// TIA Portal V20 export
FUNCTION_BLOCK "FB_Msg"   // FB84, SCL
{ S7_Optimized_Access := 'TRUE' }
// stored: MemoryReserve 100, SetENOAutomatically false
   VAR
      sSeverity : Byte;
      sMemoNumberOfActiveAlarms : DInt;
      sTON_On : TON_TIME;
      sTON_OFF { S7_SetPoint := 'True'} : TON_TIME;
      sPulseUpdateAlarms { S7_SetPoint := 'True'} : Bool;
      sRT_PulseUpdateAlarms : R_TRIG;
   END_VAR
   VAR_TEMP
      tIndex1 : Int;
      tIndex2 : Int;
      tResultByte0 : Int;
   END_VAR
   VAR CONSTANT
      MSG_SIZE : Int := 95;
   END_VAR
BEGIN
   // REGION Test
   //     FOR #tIndex := 0 TO #MSG_SIZE DO
   //         #tResultByte0 := PEEK(area := 16#84, dbNumber := 2, byteOffset := #tIndex + 554);
   //         "Db_Messages".Msg[#tIndex].ID := #tIndex;
   //         "Db_Messages".Msg[#tIndex].Number := INT_TO_DINT(#tIndex) + 70000;
   //         "Db_Messages".Msg[#tIndex].Active := #tResultByte0.%X0;
   //     END_FOR;
   // END_REGION

   REGION Format Msg
       // Mise en forme des alarmes (DB2) dans DB_FormatMsg
       FOR #tIndex1 := 0 TO 8 DO
           FOR #tIndex2 := 0 TO 7 DO
               #tResultByte0 := PEEK(area := 16#84, dbNumber := 2, byteOffset := #tIndex2 + 554 + (#tIndex1 * 8));
               "DB_FormatMsg".Msg[(#tIndex2 * 8) + (#tIndex1 * 64) + 0].Id := INT_TO_DINT((#tIndex2 * 8) + 0) + 70000 + (#tIndex1 * 100);
               "DB_FormatMsg".Msg[(#tIndex2 * 8) + (#tIndex1 * 64) + 1].Id := INT_TO_DINT((#tIndex2 * 8) + 1) + 70000 + (#tIndex1 * 100);
               "DB_FormatMsg".Msg[(#tIndex2 * 8) + (#tIndex1 * 64) + 2].Id := INT_TO_DINT((#tIndex2 * 8) + 2) + 70000 + (#tIndex1 * 100);
               "DB_FormatMsg".Msg[(#tIndex2 * 8) + (#tIndex1 * 64) + 3].Id := INT_TO_DINT((#tIndex2 * 8) + 3) + 70000 + (#tIndex1 * 100);
               "DB_FormatMsg".Msg[(#tIndex2 * 8) + (#tIndex1 * 64) + 4].Id := INT_TO_DINT((#tIndex2 * 8) + 4) + 70000 + (#tIndex1 * 100);
               "DB_FormatMsg".Msg[(#tIndex2 * 8) + (#tIndex1 * 64) + 5].Id := INT_TO_DINT((#tIndex2 * 8) + 5) + 70000 + (#tIndex1 * 100);
               "DB_FormatMsg".Msg[(#tIndex2 * 8) + (#tIndex1 * 64) + 6].Id := INT_TO_DINT((#tIndex2 * 8) + 6) + 70000 + (#tIndex1 * 100);
               "DB_FormatMsg".Msg[(#tIndex2 * 8) + (#tIndex1 * 64) + 7].Id := INT_TO_DINT((#tIndex2 * 8) + 7) + 70000 + (#tIndex1 * 100);

               "DB_FormatMsg".Msg[(#tIndex2 * 8) + (#tIndex1 * 64) + 0].Active := #tResultByte0.%X0;
               "DB_FormatMsg".Msg[(#tIndex2 * 8) + (#tIndex1 * 64) + 1].Active := #tResultByte0.%X1;
               "DB_FormatMsg".Msg[(#tIndex2 * 8) + (#tIndex1 * 64) + 2].Active := #tResultByte0.%X2;
               "DB_FormatMsg".Msg[(#tIndex2 * 8) + (#tIndex1 * 64) + 3].Active := #tResultByte0.%X3;
               "DB_FormatMsg".Msg[(#tIndex2 * 8) + (#tIndex1 * 64) + 4].Active := #tResultByte0.%X4;
               "DB_FormatMsg".Msg[(#tIndex2 * 8) + (#tIndex1 * 64) + 5].Active := #tResultByte0.%X5;
               "DB_FormatMsg".Msg[(#tIndex2 * 8) + (#tIndex1 * 64) + 6].Active := #tResultByte0.%X6;
               "DB_FormatMsg".Msg[(#tIndex2 * 8) + (#tIndex1 * 64) + 7].Active := #tResultByte0.%X7;
           END_FOR;
       END_FOR;
   END_REGION

   REGION Severity WFA A REVOIR !!
       #sSeverity := 1;
       "DB_FormatMsg".Msg[35].Severity := #sSeverity;

       "DB_FormatMsg".Msg[236].Severity := #sSeverity;

       "DB_FormatMsg".Msg[532].Severity := #sSeverity;
       "DB_FormatMsg".Msg[533].Severity := #sSeverity;
       "DB_FormatMsg".Msg[534].Severity := #sSeverity;
       "DB_FormatMsg".Msg[535].Severity := #sSeverity;
       "DB_FormatMsg".Msg[536].Severity := #sSeverity;
       "DB_FormatMsg".Msg[537].Severity := #sSeverity;
       "DB_FormatMsg".Msg[538].Severity := #sSeverity;
       "DB_FormatMsg".Msg[539].Severity := #sSeverity;
       "DB_FormatMsg".Msg[542].Severity := #sSeverity;
       "DB_FormatMsg".Msg[548].Severity := #sSeverity;
       "DB_FormatMsg".Msg[550].Severity := #sSeverity;
       "DB_FormatMsg".Msg[551].Severity := #sSeverity;

       "DB_FormatMsg".Msg[800].Severity := #sSeverity;
       "DB_FormatMsg".Msg[841].Severity := #sSeverity;

       #sSeverity := 2;
       "DB_FormatMsg".Msg[59].Severity := #sSeverity;
       "DB_FormatMsg".Msg[60].Severity := #sSeverity;
       "DB_FormatMsg".Msg[61].Severity := #sSeverity;
       "DB_FormatMsg".Msg[62].Severity := #sSeverity;

       "DB_FormatMsg".Msg[348].Severity := #sSeverity;

       "DB_FormatMsg".Msg[441].Severity := #sSeverity;
       "DB_FormatMsg".Msg[442].Severity := #sSeverity;

       "DB_FormatMsg".Msg[543].Severity := #sSeverity;

       "DB_FormatMsg".Msg[662].Severity := #sSeverity;
       "DB_FormatMsg".Msg[663].Severity := #sSeverity;

       // "DB_FormatMsg".Msg[3032].Severity := #sSeverity;
       // "DB_FormatMsg".Msg[3033].Severity := #sSeverity;
       // "DB_FormatMsg".Msg[3034].Severity := #sSeverity;
       // "DB_FormatMsg".Msg[3035].Severity := #sSeverity;
       // "DB_FormatMsg".Msg[3036].Severity := #sSeverity;
       // "DB_FormatMsg".Msg[3037].Severity := #sSeverity;
       // "DB_FormatMsg".Msg[3038].Severity := #sSeverity;
       // "DB_FormatMsg".Msg[3039].Severity := #sSeverity;
       // "DB_FormatMsg".Msg[3010].Severity := #sSeverity;
       // "DB_FormatMsg".Msg[3041].Severity := #sSeverity;
       // "DB_FormatMsg".Msg[3042].Severity := #sSeverity;
       // "DB_FormatMsg".Msg[3043].Severity := #sSeverity;
       // "DB_FormatMsg".Msg[3044].Severity := #sSeverity;
       // "DB_FormatMsg".Msg[3045].Severity := #sSeverity;
       // "DB_FormatMsg".Msg[3046].Severity := #sSeverity;
       // "DB_FormatMsg".Msg[3047].Severity := #sSeverity;


       "DB_FormatMsg".Msg[55].Severity := #sSeverity;
       "DB_FormatMsg".Msg[63].Severity := #sSeverity;

       "DB_FormatMsg".Msg[403].Severity := #sSeverity;
       "DB_FormatMsg".Msg[404].Severity := #sSeverity;
       "DB_FormatMsg".Msg[405].Severity := #sSeverity;
       "DB_FormatMsg".Msg[406].Severity := #sSeverity;
       "DB_FormatMsg".Msg[420].Severity := #sSeverity;
       "DB_FormatMsg".Msg[421].Severity := #sSeverity;
       "DB_FormatMsg".Msg[422].Severity := #sSeverity;
       "DB_FormatMsg".Msg[423].Severity := #sSeverity;

       "DB_FormatMsg".Msg[508].Severity := #sSeverity;
       "DB_FormatMsg".Msg[509].Severity := #sSeverity;
       "DB_FormatMsg".Msg[510].Severity := #sSeverity;
       "DB_FormatMsg".Msg[511].Severity := #sSeverity;
       "DB_FormatMsg".Msg[512].Severity := #sSeverity;

       "DB_FormatMsg".Msg[652].Severity := #sSeverity;
       "DB_FormatMsg".Msg[653].Severity := #sSeverity;

       "DB_FormatMsg".Msg[700].Severity := #sSeverity;
       "DB_FormatMsg".Msg[701].Severity := #sSeverity;
       "DB_FormatMsg".Msg[702].Severity := #sSeverity;
       "DB_FormatMsg".Msg[703].Severity := #sSeverity;
       "DB_FormatMsg".Msg[704].Severity := #sSeverity;
       "DB_FormatMsg".Msg[705].Severity := #sSeverity;
       "DB_FormatMsg".Msg[706].Severity := #sSeverity;
       "DB_FormatMsg".Msg[707].Severity := #sSeverity;
       "DB_FormatMsg".Msg[708].Severity := #sSeverity;
       "DB_FormatMsg".Msg[709].Severity := #sSeverity;
       "DB_FormatMsg".Msg[710].Severity := #sSeverity;
       "DB_FormatMsg".Msg[711].Severity := #sSeverity;
       "DB_FormatMsg".Msg[740].Severity := #sSeverity;
       "DB_FormatMsg".Msg[741].Severity := #sSeverity;
       "DB_FormatMsg".Msg[742].Severity := #sSeverity;
       "DB_FormatMsg".Msg[743].Severity := #sSeverity;
       "DB_FormatMsg".Msg[744].Severity := #sSeverity;
       "DB_FormatMsg".Msg[745].Severity := #sSeverity;
       "DB_FormatMsg".Msg[746].Severity := #sSeverity;
       "DB_FormatMsg".Msg[747].Severity := #sSeverity;
       "DB_FormatMsg".Msg[748].Severity := #sSeverity;
       "DB_FormatMsg".Msg[749].Severity := #sSeverity;
       "DB_FormatMsg".Msg[750].Severity := #sSeverity;
       "DB_FormatMsg".Msg[751].Severity := #sSeverity;
       "DB_FormatMsg".Msg[752].Severity := #sSeverity;
       "DB_FormatMsg".Msg[753].Severity := #sSeverity;
       "DB_FormatMsg".Msg[754].Severity := #sSeverity;
       "DB_FormatMsg".Msg[755].Severity := #sSeverity;
       "DB_FormatMsg".Msg[756].Severity := #sSeverity;
       "DB_FormatMsg".Msg[757].Severity := #sSeverity;
       "DB_FormatMsg".Msg[758].Severity := #sSeverity;
       "DB_FormatMsg".Msg[759].Severity := #sSeverity;
       "DB_FormatMsg".Msg[760].Severity := #sSeverity;
       "DB_FormatMsg".Msg[761].Severity := #sSeverity;

       // "DB_FormatMsg".Msg[3000].Severity := #sSeverity;
       // "DB_FormatMsg".Msg[3001].Severity := #sSeverity;
       // "DB_FormatMsg".Msg[3002].Severity := #sSeverity;
       // "DB_FormatMsg".Msg[3003].Severity := #sSeverity;
       // "DB_FormatMsg".Msg[3004].Severity := #sSeverity;
       // "DB_FormatMsg".Msg[3005].Severity := #sSeverity;
       // "DB_FormatMsg".Msg[3006].Severity := #sSeverity;
       // "DB_FormatMsg".Msg[3007].Severity := #sSeverity;
       // "DB_FormatMsg".Msg[3008].Severity := #sSeverity;
       // "DB_FormatMsg".Msg[3009].Severity := #sSeverity;
       // "DB_FormatMsg".Msg[3010].Severity := #sSeverity;
       // "DB_FormatMsg".Msg[3011].Severity := #sSeverity;
       // "DB_FormatMsg".Msg[3012].Severity := #sSeverity;
       // "DB_FormatMsg".Msg[3013].Severity := #sSeverity;
       // "DB_FormatMsg".Msg[3014].Severity := #sSeverity;
       // "DB_FormatMsg".Msg[3015].Severity := #sSeverity;


       #sSeverity := 3;
       "DB_FormatMsg".Msg[6].Severity := #sSeverity;
       "DB_FormatMsg".Msg[7].Severity := #sSeverity;
       "DB_FormatMsg".Msg[8].Severity := #sSeverity;

       "DB_FormatMsg".Msg[103].Severity := #sSeverity;
       "DB_FormatMsg".Msg[104].Severity := #sSeverity;
       "DB_FormatMsg".Msg[105].Severity := #sSeverity;
       "DB_FormatMsg".Msg[106].Severity := #sSeverity;
       "DB_FormatMsg".Msg[107].Severity := #sSeverity;
       "DB_FormatMsg".Msg[108].Severity := #sSeverity;
       "DB_FormatMsg".Msg[109].Severity := #sSeverity;
       "DB_FormatMsg".Msg[110].Severity := #sSeverity;
       "DB_FormatMsg".Msg[111].Severity := #sSeverity;
       "DB_FormatMsg".Msg[112].Severity := #sSeverity;
       "DB_FormatMsg".Msg[113].Severity := #sSeverity;
       "DB_FormatMsg".Msg[114].Severity := #sSeverity;
       "DB_FormatMsg".Msg[115].Severity := #sSeverity;
       "DB_FormatMsg".Msg[120].Severity := #sSeverity;

       "DB_FormatMsg".Msg[200].Severity := #sSeverity;
       "DB_FormatMsg".Msg[201].Severity := #sSeverity;
       "DB_FormatMsg".Msg[202].Severity := #sSeverity;
       "DB_FormatMsg".Msg[204].Severity := #sSeverity;
       "DB_FormatMsg".Msg[205].Severity := #sSeverity;
       "DB_FormatMsg".Msg[206].Severity := #sSeverity;
       "DB_FormatMsg".Msg[207].Severity := #sSeverity;
       "DB_FormatMsg".Msg[208].Severity := #sSeverity;
       "DB_FormatMsg".Msg[209].Severity := #sSeverity;
       "DB_FormatMsg".Msg[210].Severity := #sSeverity;
       "DB_FormatMsg".Msg[211].Severity := #sSeverity;
       "DB_FormatMsg".Msg[212].Severity := #sSeverity;
       "DB_FormatMsg".Msg[218].Severity := #sSeverity;
       "DB_FormatMsg".Msg[219].Severity := #sSeverity;
       "DB_FormatMsg".Msg[220].Severity := #sSeverity;
       "DB_FormatMsg".Msg[221].Severity := #sSeverity;
       "DB_FormatMsg".Msg[222].Severity := #sSeverity;

       "DB_FormatMsg".Msg[315].Severity := #sSeverity;
       "DB_FormatMsg".Msg[316].Severity := #sSeverity;
       "DB_FormatMsg".Msg[317].Severity := #sSeverity;
       "DB_FormatMsg".Msg[318].Severity := #sSeverity;
       "DB_FormatMsg".Msg[319].Severity := #sSeverity;
       "DB_FormatMsg".Msg[320].Severity := #sSeverity;
       "DB_FormatMsg".Msg[321].Severity := #sSeverity;
       "DB_FormatMsg".Msg[322].Severity := #sSeverity;
       "DB_FormatMsg".Msg[323].Severity := #sSeverity;
       "DB_FormatMsg".Msg[324].Severity := #sSeverity;
       "DB_FormatMsg".Msg[325].Severity := #sSeverity;
       "DB_FormatMsg".Msg[326].Severity := #sSeverity;

       "DB_FormatMsg".Msg[409].Severity := #sSeverity;
       "DB_FormatMsg".Msg[410].Severity := #sSeverity;
       "DB_FormatMsg".Msg[424].Severity := #sSeverity;
       "DB_FormatMsg".Msg[425].Severity := #sSeverity;
       "DB_FormatMsg".Msg[426].Severity := #sSeverity;
       "DB_FormatMsg".Msg[427].Severity := #sSeverity;
       "DB_FormatMsg".Msg[428].Severity := #sSeverity;
       "DB_FormatMsg".Msg[429].Severity := #sSeverity;

       "DB_FormatMsg".Msg[604].Severity := #sSeverity;
       "DB_FormatMsg".Msg[605].Severity := #sSeverity;
       "DB_FormatMsg".Msg[606].Severity := #sSeverity;
       "DB_FormatMsg".Msg[607].Severity := #sSeverity;
       "DB_FormatMsg".Msg[608].Severity := #sSeverity;
       "DB_FormatMsg".Msg[609].Severity := #sSeverity;
       "DB_FormatMsg".Msg[610].Severity := #sSeverity;
       "DB_FormatMsg".Msg[611].Severity := #sSeverity;
       "DB_FormatMsg".Msg[640].Severity := #sSeverity;
       "DB_FormatMsg".Msg[641].Severity := #sSeverity;
       "DB_FormatMsg".Msg[650].Severity := #sSeverity;
       "DB_FormatMsg".Msg[651].Severity := #sSeverity;
       "DB_FormatMsg".Msg[654].Severity := #sSeverity;
       "DB_FormatMsg".Msg[655].Severity := #sSeverity;
       "DB_FormatMsg".Msg[656].Severity := #sSeverity;
       "DB_FormatMsg".Msg[657].Severity := #sSeverity;
       "DB_FormatMsg".Msg[658].Severity := #sSeverity;
       "DB_FormatMsg".Msg[659].Severity := #sSeverity;
       "DB_FormatMsg".Msg[660].Severity := #sSeverity;
       "DB_FormatMsg".Msg[661].Severity := #sSeverity;

       "DB_FormatMsg".Msg[808].Severity := #sSeverity;
       "DB_FormatMsg".Msg[809].Severity := #sSeverity;
       "DB_FormatMsg".Msg[810].Severity := #sSeverity;
       "DB_FormatMsg".Msg[811].Severity := #sSeverity;
       "DB_FormatMsg".Msg[812].Severity := #sSeverity;
       "DB_FormatMsg".Msg[813].Severity := #sSeverity;
       "DB_FormatMsg".Msg[814].Severity := #sSeverity;
       "DB_FormatMsg".Msg[815].Severity := #sSeverity;
       "DB_FormatMsg".Msg[816].Severity := #sSeverity;
       "DB_FormatMsg".Msg[817].Severity := #sSeverity;
       "DB_FormatMsg".Msg[820].Severity := #sSeverity;
       "DB_FormatMsg".Msg[821].Severity := #sSeverity;
       "DB_FormatMsg".Msg[822].Severity := #sSeverity;
       "DB_FormatMsg".Msg[823].Severity := #sSeverity;
       "DB_FormatMsg".Msg[824].Severity := #sSeverity;

       "DB_FormatMsg".Msg[2].Severity := #sSeverity;
       "DB_FormatMsg".Msg[5].Severity := #sSeverity;

       "DB_FormatMsg".Msg[501].Severity := #sSeverity;
       "DB_FormatMsg".Msg[502].Severity := #sSeverity;

       "DB_FormatMsg".Msg[642].Severity := #sSeverity;
       "DB_FormatMsg".Msg[643].Severity := #sSeverity;
       "DB_FormatMsg".Msg[644].Severity := #sSeverity;
       "DB_FormatMsg".Msg[645].Severity := #sSeverity;
       "DB_FormatMsg".Msg[646].Severity := #sSeverity;
       "DB_FormatMsg".Msg[647].Severity := #sSeverity;
       "DB_FormatMsg".Msg[648].Severity := #sSeverity;
       "DB_FormatMsg".Msg[649].Severity := #sSeverity;

       #sSeverity := 4;
       "DB_FormatMsg".Msg[3].Severity := #sSeverity;
       "DB_FormatMsg".Msg[4].Severity := #sSeverity;

       "DB_FormatMsg".Msg[330].Severity := #sSeverity;
       "DB_FormatMsg".Msg[331].Severity := #sSeverity;

       "DB_FormatMsg".Msg[500].Severity := #sSeverity;

       "DB_FormatMsg".Msg[600].Severity := #sSeverity;
       "DB_FormatMsg".Msg[601].Severity := #sSeverity;
       "DB_FormatMsg".Msg[602].Severity := #sSeverity;
       "DB_FormatMsg".Msg[603].Severity := #sSeverity;
       "DB_FormatMsg".Msg[623].Severity := #sSeverity;
       "DB_FormatMsg".Msg[625].Severity := #sSeverity;

       "DB_FormatMsg".Msg[402].Severity := #sSeverity;
   END_REGION

   REGION Active Alarms
       // Recherche des alarmes actives dans DB_FormatMsg
       #tIndex2 := 0;
       FOR #tIndex1 := 0 TO 575 DO
           IF "DB_FormatMsg".Msg[#tIndex1].Active THEN
               "DB_ActiveAlarms".ActiveAlarms[#tIndex2].Id := "DB_FormatMsg".Msg[#tIndex1].Id;
               "DB_ActiveAlarms".ActiveAlarms[#tIndex2].Severity := "DB_FormatMsg".Msg[#tIndex1].Severity;
               #tIndex2 := #tIndex2 + 1;
           END_IF;
       END_FOR;
       "DB_ActiveAlarms".NumberOfActiveAlarms := #tIndex2;
   END_REGION

   REGION Update alarms
       // TON phase ON (5 secondes)
       #sTON_On(
                IN := #sPulseUpdateAlarms,
                PT := T#5s);

       // TON phase OFF (5 secondes)
       #sTON_OFF(
                 IN := NOT #sPulseUpdateAlarms,
                 PT := T#5s);

       IF #sTON_On.Q THEN
           #sPulseUpdateAlarms := FALSE;
       END_IF;

       IF #sTON_OFF.Q THEN
           #sPulseUpdateAlarms := TRUE;
       END_IF;

       #sRT_PulseUpdateAlarms(CLK := #sPulseUpdateAlarms);

       IF ("DB_ActiveAlarms".NumberOfActiveAlarms <> #sMemoNumberOfActiveAlarms) OR #sRT_PulseUpdateAlarms.Q THEN
           "DB_ActiveAlarms".Update := "DB_ActiveAlarms".Update + 1;
           IF "DB_ActiveAlarms".Update > 255 OR "DB_ActiveAlarms".Update < 1 THEN
               "DB_ActiveAlarms".Update := 1;
           END_IF;
       END_IF;
   END_REGION

   REGION Transfert to OPC
       "DB_OPC_Alarms".ActiveAlarms := "DB_ActiveAlarms".ActiveAlarms;
       "DB_OPC_Alarms".NumberOfActiveAlarms := "DB_ActiveAlarms".NumberOfActiveAlarms;
       "DB_OPC_Alarms".Update := "DB_ActiveAlarms".Update;
   END_REGION
END_FUNCTION_BLOCK
